INTERFACE I_AxisMoveModulo EXTENDS I_Base

METHOD MoveModulo : BOOL
VAR_INPUT
	Position	  : LREAL;
	AbortPrevious : BOOL		 := TRUE;
END_VAR
END_METHOD

END_INTERFACE

(* stored: Version 1.1.0.1, ProductVersion 3.1.4026.20
   Itf I_AxisMoveModulo: Id {3c965038-613b-4dbe-8f40-273178be4a6e}
   Method MoveModulo: Id {23992595-2597-4738-bd01-e01eeced0372} *)
